(* CoDeSys 2.3.9.59 project: abc.pro *)
(* Libraries: STANDARD.LIB *)

(* Task configuration *)
TASK Standard (PRIORITY := 0, INTERVAL := T#10ms);
	MAIN
END_TASK

(* POU MAIN, IL *)
PROGRAM MAIN
VAR
END_VAR

END_PROGRAM
